ABB RobotStudio station: Obelix2_20190228-092303.rsstn

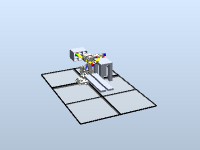
Station Obelix2 (saved by RobotStudio 6.8.8148.134)
Controller IRB_140T_6kg_0.81m
  mechanical unit ROB_1: IRB140T_6_81_C_03, 6 joints, base frame (0, 0, 0) mm
Layout (positions relative to the parent item):
  - IRB140T_6_81_C_03 [mechanism, from Robots\IRB140T_6_81_C_G_03.rslib] at (0, 0, 0) mm; joint values [-0.0127, -0.0195, 0.0068, -0.0003, 0.0389, -0.0167] (rad or m)
  - conveyor [part]
  - ManipulationTable [part]
  - conveyor_2 [part]
  - Oven_2 [part]
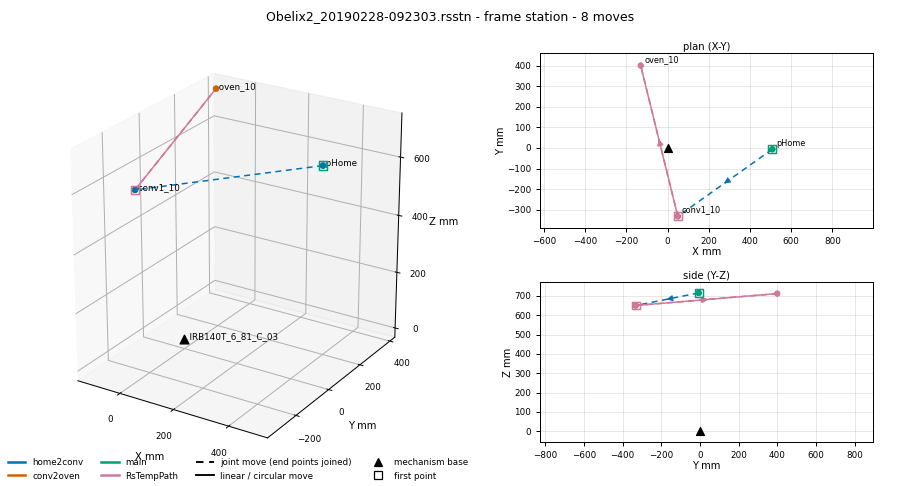
[picture p0: tool path of Obelix2_20190228-092303.rsstn in frame station, 8 of 8 moves have a stored position in this frame; points joined in program order, loops and branches not executed]
Targets, tools, work objects and paths stored in the station, written as RAPID:
! task T_ROB1
MODULE CalibData
  CONST robtarget pHome:=[[507.9,-6.43,715.02],[0.697685,-0.00154316,0.716328,-0.0103435],[-1,-1,-1,0],[9E+09,9E+09,9E+09,9E+09,9E+09,9E+09]];
  CONST robtarget conv1_10:=[[49.3280625,-331.922,650],[0,0,1,0],[0,0,0,0],[9E+09,9E+09,9E+09,9E+09,9E+09,9E+09]];
  CONST robtarget oven_10:=[[-130.719696045,400,711.666666667],[0,1,0,0],[0,0,0,0],[9E+09,9E+09,9E+09,9E+09,9E+09,9E+09]];
ENDMODULE

! task T_ROB1
MODULE Module1
  CONST robtarget man_10:=[[325,6.025878906,553],[0,-0.707106781,0.707106781,0],[0,0,0,0],[9E+09,9E+09,9E+09,9E+09,9E+09,9E+09]];
  PROC home2conv()
    MoveJ pHome,v1000,z100,tool0\WObj:=wobj0;
    MoveJ conv1_10,v1000,z100,tool0\WObj:=wobj0;
  ENDPROC
  PROC conv2oven()
    MoveJ conv1_10,v1000,fine,tool0\WObj:=wobj0;
    MoveJ oven_10,v1000,fine,tool0\WObj:=wobj0;
  ENDPROC
ENDMODULE

! task T_ROB1
MODULE ObelixMov
  PROC main()
    MoveJ pHome,v1000,fine,tool0;
    MoveJ pHome,v1000,fine,tool0;
  ENDPROC
ENDMODULE

! task T_ROB1
MODULE RsTempModule
  LOCAL CONST robtarget conv1_10:=[[49.3280625,-331.922,650],[0,0,1,0],[0,0,0,0],[9E+09,9E+09,9E+09,9E+09,9E+09,9E+09]];
  LOCAL CONST robtarget oven_10:=[[-130.719696045,400,711.666666667],[0,1,0,0],[0,0,0,0],[9E+09,9E+09,9E+09,9E+09,9E+09,9E+09]];
  PROC RsTempPath()
    MoveL conv1_10,v1000,z100,tool0\WObj:=wobj0;
    MoveL oven_10,v1000,z100,tool0\WObj:=wobj0;
  ENDPROC
ENDMODULE

